# B&R Automation Studio project MIG1 (part 12)

```c
}
void readAttribute_CoolerSens(Arc_Link_typ *arc){
	// Create a Request Message and header
	Robot_typ *robot;
	Arc_Link_Request_typ *r;
	Arc_Link_Header_typ *h;
	PendingResponse_typ *pr;

	if(!arc) return;

	pr = &arc->PendingResponse;
	robot = &arc->robot;
	r = &arc->msgOUT.request;
	h = &arc->msgOUT.header;

	// Create a UDP Request Header with all the required info
	r->TimeoutTime = 10; // 10 ms
	r->Flags = 0;
	r->Retries = 1;
	r->MessageCounter = 0;
	r->AddressingMode = 6;
	r->ConnectionID = 15;
	r->MaximumObjs = 1;
	r->ServiceID.AttributeNumber = 0x7B09;
	r->ServiceID.StateNumber = 0;
	r->ServiceID.PropertyNumber = PROPERTY_ID_VALUE;

	//The attribute for the pump status (separate from the pump command) is 0x7875, and the attribute for the flow status is 0x7B09.

	r->SourceAddress = robot->arclink.network.ModuleBaseAddress;
	r->DestinationAddress = robot->miscSetup.CoolerAddr ;// Weld Controller
	r->Service = NETWORK_SERVICE_ATTRIBUTE_READ;
	r->MaxResponseSize = 254;

	//r->OutgoingData = er.encode();
	r->RequestSize = 0; // Size

	// Data must be sent in Big Endian format
	// Create a Response header for reply
	h->Flags 		= 0x02; // Arclink Request 0b0010

	// It has to be the same as request header
	h->Sequence 	= rand();
	pr->sqReadCoolerSens = h->Sequence;
	h->LastError 	= 0;
	h->DataLength 	= ARC_LINK_REQUEST_SIZE + r->RequestSize; // This depends on
	// size of data
	// being sent
	// 6(ARcklink
	// Response size +
	// Data size)

	/* Now encode ArcLink Header and Response */
	//arc->internal.OutMsgLen = ARC_LINK_HEADER_SIZE + h->DataLength;
	arc->internal.OutMsgLen = ARC_LINK_HEADER_SIZE + h->DataLength;

	// Temp Data
	int RequestSize = r->RequestSize;

	// Swap bytes into Big Endian Format
	swapArcLinkHeaderBytes(h);
	swapArcLinkRequestBytes(r);

	memcpy(arc->internal.pOutMsg, h , ARC_LINK_HEADER_SIZE);
	memcpy(arc->internal.pOutMsg + ARC_LINK_HEADER_SIZE, r , ARC_LINK_REQUEST_SIZE);

	// Swap bytes into Big Endian Format
	//swapArcLinkHeaderBytes(h);
	//swapArcLinkRequestBytes(r);

	// Arclink Request is ready to be sent
	writeMessageToOutgoingRingBuffer(arc);

	log_event(&robot->eventlog , "Get Cooler Sens REQ");
}

void action_ConfigDataSearch_GasSol(Arc_Link_typ *arc){
	// Create a Request Message and header
	Robot_typ *robot;
	Arc_Link_Request_typ *r;
	Arc_Link_Header_typ *h;
	PendingResponse_typ *pr;

	if(!arc) return;

	pr = &arc->PendingResponse;

	robot = &arc->robot;
	r = &arc->msgOUT.request;
	h = &arc->msgOUT.header;

	// Create a UDP Request Header with all the required info
	r->TimeoutTime = 10; // 10 ms
	r->Flags = 0;
	r->Retries = 1;
	r->MessageCounter = 0;
	r->AddressingMode = 6;
	r->ConnectionID = 15;
	r->MaximumObjs = 1;
	r->ServiceID.AttributeNumber = ACTION_CONFIG_DATA_SEARCH; //Configuration Data Search ACTION
	r->ServiceID.StateNumber = 0;
	r->ServiceID.PropertyNumber = PROPERTY_ID_VALUE;

	r->SourceAddress = robot->arclink.network.ModuleBaseAddress;
	r->DestinationAddress = WELD_CONTROLLER_NETWORK_ADDRESS; //BUS_MASTER_ARCLINK_NETWORK_ADDRESS;
	r->Service = NETWORK_SERVICE_ACTION;
	r->MaxResponseSize = 254;

	//r->OutgoingData = er.encode();
	r->RequestSize = 8; //
	USINT data[8];

	/*
	Request
	1 Byte	Search Parameter Mask
	1 Byte	Group Assignment
	2 Bytes Object Class
	1 Byte	Object Instance
	1 Byte	Object Class Type
	1 Byte	Maximum
	1 Byte	Starting Network Address
*/

	data[0] = 0x4; //Mask - Attribute Class

	data[1] = 0;

	data[2] = 0; //Bytes Object Class
	//data[3] = 29; //Bytes Object Class - Cooler
	data[3] = 22; //Bytes Object Class - Remote Control object (object class ID 22)

	data[4] = 0;
	data[5] = 0;
	data[6] = 1;
	data[7] = 1;

	memcpy(arc->internal.pOutMsg + ARC_LINK_HEADER_SIZE + ARC_LINK_REQUEST_SIZE, &data[0] , r->RequestSize);

	// Data must be sent in Big Endian format
	// Create a Response header for reply
	h->Flags 		= 0x02; // Arclink Request 0b0010

	// It has to be the same as request header
	h->Sequence 	= rand();
	h->LastError 	= 0;
	h->DataLength 	= ARC_LINK_REQUEST_SIZE + r->RequestSize; // This depends on
	// size of data
	// being sent
	// 6(ARcklink
	// Response size +
	// Data size)

	/* Now encode ArcLink Header and Response */
	//arc->internal.OutMsgLen = ARC_LINK_HEADER_SIZE + h->DataLength;
	arc->internal.OutMsgLen = ARC_LINK_HEADER_SIZE + h->DataLength;

	pr->sqConfigDataSearchAction_GasSol = 	h->Sequence;

	// Temp Data
	int RequestSize = r->RequestSize;

	// Swap bytes into Big Endian Format
	swapArcLinkHeaderBytes(h);
	swapArcLinkRequestBytes(r);

	memcpy(arc->internal.pOutMsg, h , ARC_LINK_HEADER_SIZE);
	memcpy(arc->internal.pOutMsg + ARC_LINK_HEADER_SIZE, r , ARC_LINK_REQUEST_SIZE);

	// Swap bytes into Big Endian Format
	//swapArcLinkHeaderBytes(h);
	//swapArcLinkRequestBytes(r);

	// Arclink Request is ready to be sent

	writeMessageToOutgoingRingBuffer(arc);

	log_event(&robot->eventlog , "Get Cooler Adr REQ");
}

void action_ConfigDataSearch(Arc_Link_typ *arc){
	// Create a Request Message and header
	Robot_typ *robot;
	Arc_Link_Request_typ *r;
	Arc_Link_Header_typ *h;
	PendingResponse_typ *pr;

	if(!arc) return;

	pr = &arc->PendingResponse;

	robot = &arc->robot;
	r = &arc->msgOUT.request;
	h = &arc->msgOUT.header;

	// Create a UDP Request Header with all the required info
	r->TimeoutTime = 10; // 10 ms
	r->Flags = 0;
	r->Retries = 1;
	r->MessageCounter = 0;
	r->AddressingMode = 6;
	r->ConnectionID = 15;
	r->MaximumObjs = 1;
	r->ServiceID.AttributeNumber = ACTION_CONFIG_DATA_SEARCH; //Configuration Data Search ACTION
	r->ServiceID.StateNumber = 0;
	r->ServiceID.PropertyNumber = PROPERTY_ID_VALUE;

	r->SourceAddress = robot->arclink.network.ModuleBaseAddress;
	r->DestinationAddress = WELD_CONTROLLER_NETWORK_ADDRESS; //BUS_MASTER_ARCLINK_NETWORK_ADDRESS;
	r->Service = NETWORK_SERVICE_ACTION;
	r->MaxResponseSize = 254;

	//r->OutgoingData = er.encode();
	r->RequestSize = 8; //
	USINT data[8];

	/*
	Request
	1 Byte	Search Parameter Mask
	1 Byte	Group Assignment
	2 Bytes Object Class
	1 Byte	Object Instance
	1 Byte	Object Class Type
	1 Byte	Maximum
	1 Byte	Starting Network Address
*/

	data[0] = 0x4; //Mask - Attribute Class

	data[1] = 0;

	data[2] = 0; //Bytes Object Class
	data[3] = 29; //Bytes Object Class - Cooler
	//data[3] = 22; //Bytes Object Class - Remote Control object (object class ID 22)

	data[4] = 0;
	data[5] = 0;
	data[6] = 1;
	data[7] = 1;

	memcpy(arc->internal.pOutMsg + ARC_LINK_HEADER_SIZE + ARC_LINK_REQUEST_SIZE, &data[0] , r->RequestSize);

	// Data must be sent in Big Endian format
	// Create a Response header for reply
	h->Flags 		= 0x02; // Arclink Request 0b0010

	// It has to be the same as request header
	h->Sequence 	= rand();
	h->LastError 	= 0;
	h->DataLength 	= ARC_LINK_REQUEST_SIZE + r->RequestSize; // This depends on
	// size of data
	// being sent
	// 6(ARcklink
	// Response size +
	// Data size)

	/* Now encode ArcLink Header and Response */
	//arc->internal.OutMsgLen = ARC_LINK_HEADER_SIZE + h->DataLength;
	arc->internal.OutMsgLen = ARC_LINK_HEADER_SIZE + h->DataLength;

	pr->sqConfigDataSearchAction = 	h->Sequence;

	// Temp Data
	int RequestSize = r->RequestSize;

	// Swap bytes into Big Endian Format
	swapArcLinkHeaderBytes(h);
	swapArcLinkRequestBytes(r);

	memcpy(arc->internal.pOutMsg, h , ARC_LINK_HEADER_SIZE);
	memcpy(arc->internal.pOutMsg + ARC_LINK_HEADER_SIZE, r , ARC_LINK_REQUEST_SIZE);

	// Swap bytes into Big Endian Format
	//swapArcLinkHeaderBytes(h);
	//swapArcLinkRequestBytes(r);

	// Arclink Request is ready to be sent

	writeMessageToOutgoingRingBuffer(arc);

	log_event(&robot->eventlog , "Get Cooler Adr REQ");
}

void handleResponse_ReadCoolerSens(Arc_Link_typ *arc){
	Arc_Link_Response_typ 	*r; // temp reference to request
	Robot_typ 				*robot;
	USINT *data;

	if (!arc) return; // Prevent null pointer reference
	r = &arc->msgIN.response;
	robot = &arc->robot;

	DBG_OB("Received response for Cooler Search Address \r\n" );

	//Log.d(TAG, "Recevied Assign Network Address Action");

	// Copy Data if available to the Incoming data pointer
	if(r->ResponseSize > 0){
		//byte[] data = r.OutgoingData; // incominng data in Big endian format
		data = (arc->internal.pInMsg + ARC_LINK_HEADER_SIZE + ARC_LINK_RESPONSE_SIZE); // Pointer to data go back here and test
	}else{
		DBG_OB("Error: Receiving fault status with Response size \r\n");
		log_error(&robot->errorlog , "Cooler Sens Resp Fault");
		return;
	}

	//robot->miscSetup.CoolerAddr = data[0];
	//log_event(&robot->eventlog , "Got Cooler Adr RESP");

	robot->Cntrl.Fbk.coolerSens_Status = data[0];
	log_event(&robot->eventlog , "Got Cooler Sens");

}

void handleResponseReadControlParamDataAction(Arc_Link_typ *arc){
	Arc_Link_Response_typ 	*r; // temp reference to request
	Robot_typ 				*robot;
	USINT *data;

	if (!arc) return; // Prevent null pointer reference
	r = &arc->msgIN.response;
	robot = &arc->robot;

	DBG_OB("Received response -Read WC Param Data Action\r\n" );
	//log_event(&robot->eventlog , "Received Cooler Address from PS");

	//Log.d(TAG, "Recevied Assign Network Address Action");

	// Copy Data if available to the Incoming data pointer
	if(r->ResponseSize > 0){
		//byte[] data = r.OutgoingData; // incominng data in Big endian format
		data = (arc->internal.pInMsg + ARC_LINK_HEADER_SIZE + ARC_LINK_RESPONSE_SIZE); // Pointer to data go back here and test
		log_event(&robot->eventlog , "Got WC Param Data");
	}else{
		//DBG_OB("Error: Receiving fault status with Response size \r\n");
		log_error(&robot->errorlog , "Get WC Param Data Fault");
		return;
	}

	memset (&robot->Comm.CntrlParamData , 0 , sizeof(ReadControlParameterData_typ));
	memset (&robot->ResData_raw , 0 , sizeof(robot->ResData_raw));
	robot->ResDataSize = 0;

	if(r->ResponseSize == 1){ // return code

		robot->Comm.CntrlParamData.ReturnCode = *data;
	}
	else if((r->ResponseSize > 0)
		&&(r->ResponseSize < 32)){
		robot->ResDataSize = (UINT)r->ResponseSize;
		memcpy(robot->ResData_raw , data , r->ResponseSize);
	}
	else
		return;

	memcpy(&robot->Comm.CntrlParamData.MaxVal , (data+0) , 2);
	swapBytes((USINT *)&robot->Comm.CntrlParamData.MaxVal, 2);

	memcpy(&robot->Comm.CntrlParamData.MinVal , (data +2) , 2);
	swapBytes((USINT *)&robot->Comm.CntrlParamData.MinVal, 2);

	robot->Comm.CntrlParamData.UnitsCode = (USINT)*(data+4);

	robot->Comm.CntrlParamData.DecimalPlace = (USINT)*(data+5);
	memcpy(robot->Comm.CntrlParamData.Name ,  data+6 , 17);
	//swapBytes(robot->Comm.CntrlParamData.Name, 17);

}

void handleResponseConfigDataSearchAction_GasSol(Arc_Link_typ *arc){
	Arc_Link_Response_typ 	*r; // temp reference to request
	Robot_typ 				*robot;
	USINT *data;

	if (!arc) return; // Prevent null pointer reference
	r = &arc->msgIN.response;
	robot = &arc->robot;

	DBG_OB("Received response for Cooler Search Address \r\n" );
	//log_event(&robot->eventlog , "Received Cooler Address from PS");

	//Log.d(TAG, "Recevied Assign Network Address Action");

	// Copy Data if available to the Incoming data pointer
	if(r->ResponseSize > 0){
		//byte[] data = r.OutgoingData; // incominng data in Big endian format
		data = (arc->internal.pInMsg + ARC_LINK_HEADER_SIZE + ARC_LINK_RESPONSE_SIZE); // Pointer to data go back here and test
	}else{
		DBG_OB("Error: Receiving fault status with Response size \r\n");
		log_error(&robot->errorlog , "Gas Sol Addr Fault");
		return;
	}

	robot->miscSetup.GasSolAddr = data[0];
	log_event(&robot->eventlog , "Got Gas Sol Adr RESP");

}

void handleResponseConfigDataSearchAction(Arc_Link_typ *arc){
	Arc_Link_Response_typ 	*r; // temp reference to request
	Robot_typ 				*robot;
	USINT *data;

	if (!arc) return; // Prevent null pointer reference
	r = &arc->msgIN.response;
	robot = &arc->robot;

	DBG_OB("Received response for Cooler Search Address \r\n" );
	//log_event(&robot->eventlog , "Received Cooler Address from PS");

	//Log.d(TAG, "Recevied Assign Network Address Action");

	// Copy Data if available to the Incoming data pointer
	if(r->ResponseSize > 0){
		//byte[] data = r.OutgoingData; // incominng data in Big endian format
		data = (arc->internal.pInMsg + ARC_LINK_HEADER_SIZE + ARC_LINK_RESPONSE_SIZE); // Pointer to data go back here and test
	}else{
		DBG_OB("Error: Receiving fault status with Response size \r\n");
		log_error(&robot->errorlog , "Cooler Addr Fault");
		return;
	}

	robot->miscSetup.CoolerAddr = data[0];
	log_event(&robot->eventlog , "Got Cooler Adr RESP");

}

/*
	Error Logger by Obed Rev 1.0
*/
void log_error(Log_typ* err, char* msg){
	if(!err) return;

	// Healthy Inialization
	if(!err->pLog){
		err->pLog = &err->log;
	}

	memmove((void *)(err->pLog + LOG_MAX_LENGTH), (void *)err->pLog, (LOG_MAX_LENGTH * (LOG_MAX_LINE - 1) ));
	memmove( (void *)(err->pLog), (void *)msg, (LOG_MAX_LENGTH) );
}

void log_event(Log_typ* event, char* msg){
	if(!event) return;

	// Healthy Inialization
	if(!event->pLog){
		event->pLog = &event->log;
	}

	memmove((void *)(event->pLog + LOG_MAX_LENGTH), (void *)event->pLog, (LOG_MAX_LENGTH * (LOG_MAX_LINE - 1) ));
	memmove( (void *)(event->pLog), (void *)msg, (LOG_MAX_LENGTH) );
}
```

### Robot.c
```c
/*
 * Handler.c
 *
 *  Created on: May 18, 2017
 *      Author: Obed Bardales
 */
#ifndef _ROBOT_C
#define _ROBOT_C

/* Handle Robot Cyclic Operations */
void handleRobotCyclicOps(Arc_Link_typ *arc){
	if(!arc) return;

	// Handle Mr.Robot interface
	handleRobotInterface(arc);

	// "The difference is not one thing, it's everything!"
}

/* Get Network Configuration from Robot */
void getNetworkConfigurationAttribute(Arc_Link_typ *arc, USINT *ResponseData){
	Arc_Link_Request_typ *req;
	Arc_Link_Response_typ *r;
	Robot_typ *robot;
	ServiceID_typ *serviceID;
	ArcLinkObject_typ *arclink;
	USINT data[10]; // Temp Data place holder
	UINT txtlength; // text length

	if(!arc) return;
	if(!ResponseData) return;

	robot = &arc->robot; // Reference to Robot
	req = &arc->msgIN.request;
	serviceID = &req->ServiceID;
	r = &arc->msgOUT.response;
	arclink = &robot->arclink;
	int dataSize = req->MaxResponseSize;

	/* Attribute Number */
	switch (serviceID->AttributeNumber) {

		case VENDOR_ID: /* 0 */
			// MaxDataSize = 2
			// Big Endian Format

			data[0] = (USINT) (arclink->network.VendorID >> 8);
			data[1] = (USINT) (arclink->network.VendorID >> 0);
			memcpy(ResponseData, data, 2);
			r->ResponseSize = 2;

			return;

		case CLASS_ID: /* 4 */
			// MaxDataSize = 2
			// Big Endian Format
			data[0] = (USINT) (arclink->network.ClassID >> 8);
			data[1] = (USINT) (arclink->network.ClassID >> 0);
			memcpy(ResponseData, data, 2);
			r->ResponseSize = 2;
			return;

		case CLASS_TYPE: /* 7 */
			// MaxDataSize = 2
			// Big Endian Format
			data[0] = (USINT) (arclink->network.ClassType >> 0);
			memcpy(ResponseData, data, 1);
			r->ResponseSize = 1;
			return;

		case GROUP_ASSIGNMENTS: /* 10 */
			// MaxDataSize = 2
			// Big Endian Format
			data[0] = (USINT) (arclink->network.GroupAssignments >> 0);
			memcpy(ResponseData, data, 1);
			r->ResponseSize = 1;
			return;

		case INSTANCE_ASSIGNMENTS: /* 11 */
			// MaxDataSize = 2
			// Big Endian Format
			data[0] = (USINT) (arclink->network.InstanceAssignments >> 0);
			memcpy(ResponseData, data, 1);
			r->ResponseSize = 1;
			return;

		case FAULT_STATUS: /* 14 */
			// MaxDataSize = 2
			// Big Endian Format
			data[0] = (USINT) (arclink->network.FaultStatus >> 0);
			memcpy(ResponseData, data, 1);
			r->ResponseSize = 1;
			return;

		case SILICON_SERIAL_NUMBER: /* 16 */
			// MaxDataSize = 2
			// Big Endian Format
			data[0] = (USINT) (arclink->network.SiliconSerialNumber >> 8);
			data[1] = (USINT) (arclink->network.SiliconSerialNumber >> 0);
			memcpy(ResponseData, data, 2);
			r->ResponseSize = 2;
			return;

		case NUMBER_OF_EMBEDDED_OBJECTS: /* 17 */
			// MaxDataSize = 2
			// Big Endian Format
			data[0] = (USINT) (arclink->network.NumberofEmbeddedObjects >> 0);
			memcpy(ResponseData, data, 1);
			r->ResponseSize = 1;
			return;

		case SOFTWARE_VERSION: /* 19 */
			// MaxDataSize = 64
			// Big Endian Format
			txtlength = strlen(arclink->network.SoftwareVersion);
			// Swap Bytes before sendSuccesfullWriteAttributeConfirmation
			//swapBytes(arclink->network.SoftwareVersion, txtlength);
			memcpy(ResponseData, arclink->network.SoftwareVersion, txtlength);
			//swapBytes(arclink->network.SoftwareVersion, txtlength);
			r->ResponseSize = txtlength;
			return;

		case BOOTSTRAP: /* 24 */
			// MaxDataSize = 2
			// Big Endian Format
			data[0] = (USINT) (arclink->network.Bootstrap >> 0);
			memcpy(ResponseData, data, 1);
			r->ResponseSize = 1;
			return;

		case PAIRED_ITEMS_COUNT: /* 50 */
			// MaxDataSize = 2
			// Big Endia Format
			data[0] = (USINT) (arclink->network.PairedItemsCount >> 8);
			data[1] = (USINT) (arclink->network.PairedItemsCount >> 0);
			memcpy(ResponseData, data, 2);
			r->ResponseSize = 2;
			return;
	}
}

/* Write Network Configuration Attribute */
BOOL writeNetworkConfigurationAttribute(Arc_Link_typ *arc){

	BOOL success = 1;

	UINT *data;

	Arc_Link_Request_typ *req;
	ServiceID_typ *serviceID;
	Robot_typ *robot;
	ArcLinkObject_typ *arclink;
	if(!arc) return;

	req = &arc->msgIN.request;
	serviceID = &req->ServiceID;
	robot = &arc->robot;
	arclink = &robot->arclink;

	DBG("Inside writeNetworkConfigurationAttribute \r\n" );
	//Log.d(TAG, "Recevied Assign Network Address Action");

	// Copy Data if available to the Incoming data pointer
	if(req->RequestSize > 0){
	//byte[] data = r.OutgoingData; // incominng data in Big endian format
		data = (arc->internal.pInMsg + ARC_LINK_HEADER_SIZE + ARC_LINK_REQUEST_SIZE); // Pointer to data
	}else{
		DBG("Error: writeNetworkConfigurationAttribute, Error with Request size\r\n" );
		return;
	}

	/* Attribute Number */
	switch (serviceID->AttributeNumber) {

	// Currently Supported Attributes by the Robot
	case RESET:
		arclink->network.Reset = *(data + 0);//data[0]; // Size is typically 1 byte
		arclink->network.BusAvailable = 0; // Robot must enter to unmapped state
		robot->isMapping = 0;
		robot->isMapped = 0;
		robot->Cntrl.Fbk.Status &= ~ArcLink_Mapped;
		robot->Cntrl.Fbk.Status &= ~ArcLink_Mapping;
		robot->isMiscSetupOneShot = 0;
		DBG("Setting Robot to Unmapped state\r\n" );
		break;

	case GROUP_ASSIGNMENTS:
		arclink->network.GroupAssignments = *(data + 0);///data[0]; // Size is typically 1
													// byte

		break;

	case INSTANCE_ASSIGNMENTS:
		arclink->network.InstanceAssignments = *(data + 0);///data[0]; // Size is typically
														// 1 byte
		break;

	case BUS_AVAILABLE:
		arclink->network.BusAvailable = *(data + 0); //data[0]; // Size is typically 1 byte
		robot->isMapping 	= 0;
		robot->isMapped 	= 1;
		robot->Cntrl.Fbk.Status |= ArcLink_Mapped;
		robot->Cntrl.Fbk.Status &= ~ArcLink_Mapping;
		DBG("Robot was mapped succesfully Świetny programista! \r\n" );
		log_event(&robot->eventlog , "Arc Link Mapped");
		break;

	}

	return success; // Whether Attribute was written succesfully

}

void handleRobotInterface(Arc_Link_typ *arc){

	Robot_typ *robot;
	Robot_Intrf_typ *intrf;
	if(!arc) return;

	robot = &arc->robot;
	intrf = &robot->Intrf;

	// Robot must be Mapped with WeldController
	if(!robot->isMapped) return;

	//  Handle state changes from outside and provide feedback

	handleRobotCntrl(arc);
	error_status_handler(arc);
	ArcLink_Timer(arc);
	/////////

	// Handle xCMD
	switch(intrf->xCMD) {
		/* Turn Power Supply ON */
		case ROBOT_CMD_PS_ON:
			writeOutputOnCommand(arc);
			DBG("Robot commanded Power Supply ON! \r\n" );
			log_event(&robot->eventlog , "PS ON Cmd");
			break;

		/* Turn Power Supply OFF */
		case ROBOT_CMD_PS_OFF:
			writeOutputOffCommand(arc);
			DBG("Robot commanded Power Supply OFF! \r\n" );
			log_event(&robot->eventlog , "PS OFF Cmd");
			break;

		/* Set Controls Action Request */
		case ROBOT_SET_CONTROLS:
			createSetControlsAction(arc);
			DBG("Robot sent Set Controls Action Request! \r\n" );
			break;

		case ROBOT_CMD_COOLER_ON:
			writeOutputCoolerOnCommand(arc);
			DBG("Robot commanded Cooler ON! \r\n" );

		break;

		case ROBOT_CMD_COOLER_OFF:
			writeOutputCoolerOffCommand(arc);
			DBG("Robot commanded Cooler OFF! \r\n" );

		break;

		case ROBOT_CMD_SEARCH_COOLER_ADR:
			action_ConfigDataSearch(arc);
			DBG("commanded Get Cooler Adr! \r\n" );
		break;

		case ROBOT_READ_COOLER_SENS:
			readAttribute_CoolerSens(arc);
			DBG("commanded Get Cooler Sens! \r\n" );
		break;

		case ROBOT_READ_WC_PARAM_DATA:
			createReadCntrlParamDataAction(arc);
			DBG("commanded Read WC Param Data! \r\n" );
		break;

		case ROBOT_CMD_SEARCH_GAS_SOL_ADR:
			action_ConfigDataSearch_GasSol(arc);
			DBG("commanded Get Gas Sol  Adr! \r\n" );
		break;

		case ROBOT_CMD_GAS_SOL_ENABLE: // Make  Gas Sol “Manual Valve”

			writeOutputGasEnableCommand(arc);
			DBG("Robot commanded Gas Enable\r\n" );

		break;

		case ROBOT_CMD_GAS_SOL_ON: // Turn On Gas Sol

			writeOutputGasOnCommand(arc);
			DBG("Robot commanded Gas ON\r\n" );

		break;

		case ROBOT_CMD_GAS_SOL_OFF:	// Turn Off Gas Sol

			writeOutputGasOffCommand(arc);
			DBG("Robot commanded Gas OFF\r\n" );

		break;

	}

	// Clear xCMD
	if (intrf->xCMD > 0) intrf->xCMD = 0;

}

void handleRobotCntrl(Arc_Link_typ *arc){

	Robot_typ *robot;
	Robot_Intrf_typ *intrf;
	if(!arc) return;

	robot = &arc->robot;
	intrf = &robot->Intrf;

	//*************** CMD  *****************************/
	//**************Highest priority CMD****************//
	if(robot->Cntrl.Cmd.COOLER && !robot->Cntrl.Int._COOLER){

		intrf->xCMD = ROBOT_CMD_COOLER_ON;
		robot->Cntrl.Int._COOLER  = robot->Cntrl.Cmd.COOLER;

	}
	else if(robot->Cntrl.Cmd.RUN != robot->Cntrl.Int._RUN){

		if(robot->Cntrl.Cmd.RUN)
			intrf->xCMD = ROBOT_CMD_PS_ON;
		else
			intrf->xCMD = ROBOT_CMD_PS_OFF;

		robot->Cntrl.Int._RUN  = robot->Cntrl.Cmd.RUN;
	}
	else if(!robot->Cntrl.Cmd.COOLER && robot->Cntrl.Int._COOLER){

		intrf->xCMD = ROBOT_CMD_COOLER_OFF;
		robot->Cntrl.Int._COOLER  = robot->Cntrl.Cmd.COOLER;

	}
	//robot->Cntrl.Int._RUN  = robot->Cntrl.Cmd.RUN;
	//robot->Cntrl.Int._COOLER  = robot->Cntrl.Cmd.COOLER;

	//********************************************************//

	if(!intrf->xCMD){

		/*
		1 Byte	Parameter Mask
		2 Bytes	Weld Mode 	If parameter mask bit 0 set.
		2 Bytes	Work-point	If parameter mask bit 1 set.
		2 Bytes	Trim	If parameter mask bit 2 set.
		2 Bytes	Wave-Control 1	If parameter mask bit 3 set.
		2 Bytes	Wave-Control 2	If parameter mask bit 4 set.
		2 Bytes	Wave-Control 3	If parameter mask bit 5 set.
		2 Bytes	Wave-Control 4	If parameter mask bit 6 set.
		*/

		switch(robot->Cntrl.Cmd.Mode){

			case 3:

				if((robot->Cntrl.Cmd.Mode != robot->Cntrl.Int._Mode )
					|| (robot->Cntrl.Cmd.AmpSP != robot->Cntrl.Int._AmpSP )
					|| (robot->Cntrl.Cmd.BckAmpSP != robot->Cntrl.Int._BckAmpSP )
					|| (robot->Cntrl.Cmd.PulseFreq != robot->Cntrl.Int._PulseFreq )
					|| (robot->Cntrl.Cmd.PulseWidth != robot->Cntrl.Int._PulseWidth )){

					robot->wc.setup.ctrlParam.ParameterMask = 0x23; // 0b0100011; // change accordingly for Mode 3
					UINT *mode 	= &robot->Cntrl.Cmd.Mode; // Mode
					UINT ampSP = (UINT)robot->Cntrl.Cmd.AmpSP; //amps
					robot->wc.setup.ctrlParam.WeldMode = *mode;
					robot->wc.setup.ctrlParam.WorkPoint = ampSP;
					robot->wc.setup.ctrlParam.WaveControl3 = 1; // Hot pulse. Need info from Lincoln

					// This command write Controls Parameter into Power Supply
					intrf->xCMD = ROBOT_SET_CONTROLS;

				}

				robot->Cntrl.Int._Mode 			= robot->Cntrl.Cmd.Mode;
				robot->Cntrl.Int._AmpSP 		= robot->Cntrl.Cmd.AmpSP;
				robot->Cntrl.Int._BckAmpSP 		= robot->Cntrl.Cmd.BckAmpSP;
				robot->Cntrl.Int._PulseFreq 	= robot->Cntrl.Cmd.PulseFreq;
				robot->Cntrl.Int._PulseWidth 	= robot->Cntrl.Cmd.PulseWidth;

			break;

			case 5:

				if((robot->Cntrl.Cmd.Mode != robot->Cntrl.Int._Mode )
					|| (robot->Cntrl.Cmd.Volts != robot->Cntrl.Int._Volts )
					|| (robot->Cntrl.Cmd.Pinch != robot->Cntrl.Int._Pinch )
					){

					robot->wc.setup.ctrlParam.ParameterMask = 0x0D; // 0b0001011; // change accordingly for Mode 5
					UINT *mode 	= &robot->Cntrl.Cmd.Mode; // Mode
					UINT VoltsSP = (UINT)(robot->Cntrl.Cmd.Volts * 10); //Volts
					robot->wc.setup.ctrlParam.WeldMode = *mode;
					robot->wc.setup.ctrlParam.WorkPoint = VoltsSP;
					robot->wc.setup.ctrlParam.WaveControl1 = (UINT)(robot->Cntrl.Cmd.Pinch * 10);

					// This command write Controls Parameter into Power Supply
					intrf->xCMD = ROBOT_SET_CONTROLS;

				}

				robot->Cntrl.Int._Mode 			= robot->Cntrl.Cmd.Mode;
				robot->Cntrl.Int._Volts 		= robot->Cntrl.Cmd.Volts;
				robot->Cntrl.Int._Pinch 		= robot->Cntrl.Cmd.Pinch;

			break;

			case 21:

				if((robot->Cntrl.Cmd.Mode != robot->Cntrl.Int._Mode )
					|| (robot->Cntrl.Cmd.WFS != robot->Cntrl.Int._WFS)
					|| (robot->Cntrl.Cmd.Volts != robot->Cntrl.Int._Volts )
					|| (robot->Cntrl.Cmd.Pinch != robot->Cntrl.Int._Pinch )
					|| robot->Cntrl.Cmd.SendParam
					){

					robot->Cntrl.Cmd.SendParam = 0;

					robot->wc.setup.ctrlParam.ParameterMask = 0x0F; // 0b0001111; // change accordingly for Mode 5
					UINT *mode 	= &robot->Cntrl.Cmd.Mode; // Mode
					UINT WFS_SP = (UINT)(robot->Cntrl.Cmd.WFS * 1); //WF
					UINT VoltsSP = (UINT)(robot->Cntrl.Cmd.Volts * 10); //Volts
					UINT PinchSP = (UINT)(robot->Cntrl.Cmd.Pinch * 10); //Pinch

					if(robot->Cntrl.Cmd.Development)
						robot->wc.setup.ctrlParam.WeldMode = 0;
					else
						robot->wc.setup.ctrlParam.WeldMode = *mode;

					robot->wc.setup.ctrlParam.WorkPoint = WFS_SP;
					robot->wc.setup.ctrlParam.Trim = VoltsSP;
					robot->wc.setup.ctrlParam.WaveControl1 = PinchSP;

					// This command write Controls Parameter into Power Supply
					intrf->xCMD = ROBOT_SET_CONTROLS;

					robot->Cntrl.Int._Mode 			= robot->Cntrl.Cmd.Mode;
					robot->Cntrl.Int._WFS 			= robot->Cntrl.Cmd.WFS;
					robot->Cntrl.Int._Volts 		= robot->Cntrl.Cmd.Volts;
					robot->Cntrl.Int._Pinch 		= robot->Cntrl.Cmd.Pinch;

				}

			break;

			case 22:

				if((robot->Cntrl.Cmd.Mode != robot->Cntrl.Int._Mode )
					|| (robot->Cntrl.Cmd.WFS != robot->Cntrl.Int._WFS)
					|| (robot->Cntrl.Cmd.Trim != robot->Cntrl.Int._Trim )
					|| (robot->Cntrl.Cmd.UltimArc != robot->Cntrl.Int._UltimArc )
					|| robot->Cntrl.Cmd.SendParam
					){

					robot->Cntrl.Cmd.SendParam = 0;

					robot->wc.setup.ctrlParam.ParameterMask = 0x0F; // 0b0001111; // change accordingly for Mode 5
					UINT *mode 	= &robot->Cntrl.Cmd.Mode; // Mode
					UINT WFS_SP = (UINT)(robot->Cntrl.Cmd.WFS * 1); // WF
					UINT TrimSP = (UINT)(robot->Cntrl.Cmd.Trim * 100); // Trim
					UINT UltimArcSP = (UINT)(robot->Cntrl.Cmd.UltimArc * 10); //Pinch

					if(robot->Cntrl.Cmd.Development)
						robot->wc.setup.ctrlParam.WeldMode = 0;
					else
						robot->wc.setup.ctrlParam.WeldMode = *mode;

					robot->wc.setup.ctrlParam.WorkPoint = WFS_SP;
					robot->wc.setup.ctrlParam.Trim = TrimSP;
					robot->wc.setup.ctrlParam.WaveControl1 = UltimArcSP;

					// This command write Controls Parameter into Power Supply
					intrf->xCMD = ROBOT_SET_CONTROLS;

					robot->Cntrl.Int._Mode 			= robot->Cntrl.Cmd.Mode;
					robot->Cntrl.Int._WFS 			= robot->Cntrl.Cmd.WFS;
					robot->Cntrl.Int._Trim 			= robot->Cntrl.Cmd.Trim;
					robot->Cntrl.Int._UltimArc 		= robot->Cntrl.Cmd.UltimArc;

				}

			break;

			case 160:
			case 161:
			case 162:
			case 163:
			case 164:
			case 165:
			case 166:
			case 167:

				if((robot->Cntrl.Cmd.Mode != robot->Cntrl.Int._Mode )
					|| (robot->Cntrl.Cmd.Volts != robot->Cntrl.Int._Volts )
					//|| (robot->Cntrl.Cmd.Pinch != robot->Cntrl.Int._Pinch )
					){

					robot->wc.setup.ctrlParam.ParameterMask = 0x03; // 0b0000011; // Volts and WaveCntr 1

					//robot->wc.setup.ctrlParam.ParameterMask = 0x01; // Only Volts

					UINT *mode 	= &robot->Cntrl.Cmd.Mode; // Mode
					UINT VoltsSP = (UINT)(robot->Cntrl.Cmd.Volts * 10); // Volts
					robot->wc.setup.ctrlParam.WeldMode = *mode;
					robot->wc.setup.ctrlParam.WorkPoint = VoltsSP;
					//robot->wc.setup.ctrlParam.WaveControl1 = (UINT)(robot->Cntrl.Cmd.Pinch * 10);
					robot->wc.setup.ctrlParam.WaveControl1 = 0;

					// This command write Controls Parameter into Power Supply
					intrf->xCMD = ROBOT_SET_CONTROLS;

				}

				robot->Cntrl.Int._Mode 			= robot->Cntrl.Cmd.Mode;
				robot->Cntrl.Int._Volts 		= robot->Cntrl.Cmd.Volts;
				//robot->Cntrl.Int._Pinch 		= robot->Cntrl.Cmd.Pinch;

			break;

			case 170:

				if((robot->Cntrl.Cmd.Mode != robot->Cntrl.Int._Mode )
					|| (robot->Cntrl.Cmd.WFS != robot->Cntrl.Int._WFS)
					|| (robot->Cntrl.Cmd.Volts != robot->Cntrl.Int._Volts )
					|| (robot->Cntrl.Cmd.UltimArc != robot->Cntrl.Int._UltimArc )
					|| robot->Cntrl.Cmd.SendParam
					){

					robot->Cntrl.Cmd.SendParam = 0;

					robot->wc.setup.ctrlParam.ParameterMask = 0x0F; // 0b0001111; // change accordingly for Mode 5
					UINT *mode 	= &robot->Cntrl.Cmd.Mode; // Mode
					UINT WFS_SP = (UINT)(robot->Cntrl.Cmd.WFS * 1); //WF
					UINT VoltsSP = (UINT)(robot->Cntrl.Cmd.Volts * 10); //Volts
					UINT UltimArcSP = (UINT)(robot->Cntrl.Cmd.UltimArc * 10); //UltimArc

					if(robot->Cntrl.Cmd.Development)
						robot->wc.setup.ctrlParam.WeldMode = 0;
					else
						robot->wc.setup.ctrlParam.WeldMode = *mode;

					robot->wc.setup.ctrlParam.WorkPoint = WFS_SP;
					robot->wc.setup.ctrlParam.Trim = VoltsSP;
					robot->wc.setup.ctrlParam.WaveControl1 = UltimArcSP;

					// This command write Controls Parameter into Power Supply
					intrf->xCMD = ROBOT_SET_CONTROLS;

					robot->Cntrl.Int._Mode 			= robot->Cntrl.Cmd.Mode;
					robot->Cntrl.Int._WFS 			= robot->Cntrl.Cmd.WFS;
					robot->Cntrl.Int._Volts 		= robot->Cntrl.Cmd.Volts;
					robot->Cntrl.Int._UltimArc 		= robot->Cntrl.Cmd.UltimArc;

				}

			break;

			case 200:  // Calibration Current

				if((robot->Cntrl.Cmd.Mode != robot->Cntrl.Int._Mode )
					|| (robot->Cntrl.Cmd.AmpSP != robot->Cntrl.Int._AmpSP )
					){

					robot->wc.setup.ctrlParam.ParameterMask = 0x03; // 0b0000011; // change accordingly for Mode 200
					UINT *mode 	= &robot->Cntrl.Cmd.Mode; // Mode
					UINT AmpSP = (UINT)(robot->Cntrl.Cmd.AmpSP * 1); //amps
					robot->wc.setup.ctrlParam.WeldMode = *mode;
					robot->wc.setup.ctrlParam.WorkPoint = AmpSP;

					// This command write Controls Parameter into Power Supply
					intrf->xCMD = ROBOT_SET_CONTROLS;

				}

				robot->Cntrl.Int._Mode 			= robot->Cntrl.Cmd.Mode;
				robot->Cntrl.Int._AmpSP 		= robot->Cntrl.Cmd.AmpSP;

			break;

		}

	}
	//********************************************************//

	//*****************Lowest Priority CMD ********************//
	if(!intrf->xCMD){
		if(robot->Cntrl.Cmd.RST != robot->Cntrl.Int._RST){

			robot->Cntrl.Fbk.Status = 0;
			robot->miscSetup.state = 0; //reset misc state machine state
			robot->miscSetup.CoolerAddr = 0;
			robot->isMapping = 0;
			robot->isMapped = 0;	    //clear flag, set to unmapped status, stop timer
			robot->isMiscSetupOneShot = 0;
			robot->Comm.ArcComTimer.IN = 0;
			robot->Comm.StopRespondHeartBeat = 1; //halt heartbeat,force master to send out RESET request

		}
		robot->Cntrl.Int._RST 			= robot->Cntrl.Cmd.RST;

	}

	//*************** FEEDBACK  *****************************/

	robot->Cntrl.Fbk.curArcVolt = robot->wc.data.telemetry.fVoltage;
	robot->Cntrl.Fbk.curArcAmp  = robot->wc.data.telemetry.fCurrent;
	//robot->Cntrl.Fbk.Error      =  ???????
	//robot->Cntrl.Fbk.Status      =  ???????

	//********************************************************//

	return;

}

void error_status_handler(Arc_Link_typ *arc)
{

	Robot_typ *robot;
	if(!arc) return;

	robot = &arc->robot;

	// System is ready when mapped, ready status from PS is set and Arc Link Active, could add no system fault here
	if ((robot->isReady) && (robot->isMapped) && (robot->Comm.ArcLinkActive) && !robot->Cntrl.Fbk.Error)
	{
		robot->Cntrl.Fbk.Status |= PS_Ready;
//		log_event(&robot->eventlog , "Power supply is ready");
	}

	else
		robot->Cntrl.Fbk.Status &= ~PS_Ready;

	/*
	if ((robot->Cntrl.Fbk.Error >> 1 & 0x0001) || (robot->Cntrl.Fbk.Error >> 2 & 0x0001))  //either system fault from PS or network error will generate fault condition
		robot->Cntrl.Fbk.Error |= PS_Error_Present;
	else
		robot->Cntrl.Fbk.Error &= ~PS_Error_Present;
	*/
}
void ArcLink_Timer(Arc_Link_typ *arc){
//
	Robot_typ *robot;
	if(!arc) return;

	robot = &arc->robot;

	robot->Comm.PT = 2000; // 2s  timeout

	robot->Comm.CoolerSensPull_PT = 500; // 0.5s  timer

    robot->Comm.ArcComTimer.PT = robot->Comm.PT;

	if (robot->Comm.HeartBeat_Received && (robot->Comm.ArcComTimer.ET > 0)) //everytime got heartbeat, reset timer, to prevent trigger timeout
	    robot->Comm.ArcComTimer.IN = 0;

	else if (robot->Comm.HeartBeat_Received && (robot->Comm.ArcComTimer.ET == 0)){ //start timer, reset heartbeat flag
		if (robot->isMapped){  //
			robot->Comm.ArcComTimer.IN = 1;
		}
		if (robot->Comm.ClearError)    // clear error once getting connectivity from PS
		{
			robot->Comm.ClearError = 0;
			robot->Cntrl.Fbk.Error = 0;
			log_event(&robot->eventlog , "Network is active");
		}
		robot->Comm.HeartBeat_Received = 0;   //reset flag to start watchdog

	}

	TON(&robot->Comm.ArcComTimer);  //2 seconds Watchdog

    if (!robot->Comm.ArcComTimer.Q)
	robot->Comm.ArcLinkActive = 1;  // 1 Active
	else
	robot->Comm.ArcLinkActive = 0;	//timeout

	if (!robot->Comm.ArcLinkActive)
	{
		DBG_OB("Arc Link Disconnected\r\n");
		robot->Cntrl.Fbk.Error |= ArcLink_Com_Failed;
		robot->Cntrl.Fbk.Status = 0;
		robot->isMapping = 0;
		robot->isMapped = 0;	    //clear flag, set to unmapped status, stop timer
		robot->isMiscSetupOneShot = 0;
		robot->Comm.ArcComTimer.IN = 0;
		robot->Comm.ClearError = 1;	 //set flag when getting communication back, reset error
		log_event(&robot->eventlog , "Network is down");
	}
	else if (robot->isMapped)
	{
	/*	DBG_OB("Arc Link Connected\r\n"); */
		robot->Cntrl.Fbk.Error &= ~ArcLink_Com_Failed;
		robot->Cntrl.Fbk.Status |= ArcLink_Active;

	}

	// Pull Cooler Sens Status

	if((robot->miscSetup.CoolerAddr > 0)
		&& (robot->Comm.CoolerSensPull_PT > 0)){

		robot->Comm.CoolerSensPullTimer.PT = robot->Comm.CoolerSensPull_PT;

		if(robot->isMapped && robot->Comm.ArcLinkActive){

			if(!robot->Comm.CoolerSensPullTimer.IN){
				readAttribute_CoolerSens(arc);
				DBG("commanded Get Cooler Sens! \r\n" );
				robot->Comm.CoolerSensPullTimer.IN = 1;
				//TON(&robot->Comm.CoolerSensPullTimer);
			}
			else if(robot->Comm.CoolerSensPullTimer.Q){

				robot->Comm.CoolerSensPullTimer.IN = 0;
				//TON(&robot->Comm.CoolerSensPullTimer);

			}
			//else
				//TON(&robot->Comm.CoolerSensPullTimer);

		}

		TON(&robot->Comm.CoolerSensPullTimer);
	}

}
#endif /* _ROBOT_C */
```

### libUDP.c
```c
#ifdef _DEFAULT_INCLUDES
	#include <AsDefault.h>
#endif

/*
B&R components:
===============================================================================
*/
#include <bur/plc.h>
#include <bur/plctypes.h>

//void _NewDataSend(UDP_typ2* udp);

///////////////////////////////////////////////////////////////////////

 signed char Udp_cyclic(UDP_typ2* udp){

 	switch(udp->internal.step){

		case 0:

			udp->listener.oStatus.error_number = 0;
			udp->listener.oStatus.error = 0;
			udp->listener.oStatus.ready = 0;

			udp->send.oStatus.error_number = 0;
			udp->send.oStatus.error = 0;
			udp->send.oStatus.ready = 0;

			if(udp->listener_config.buffer && (udp->listener_config.bufferSize > 0)){

				if(udp->internal.UdpOpen_0.ident){ // CLose existing connection on start

					UdpClose(&udp->internal.UdpClose_0);  //Call the Function

					if(udp->internal.UdpClose_0.status == ERR_OK) //
						udp->internal.step = 1;

					else if (udp->internal.UdpClose_0.status == ERR_FUB_BUSY){} //UdpSend not finished -> redo

					else{  //Error

						udp->listener.oStatus.error_number = udp->internal.UdpClose_0.status;
						udp->listener.oStatus.error = 1;
						udp->listener.oStatus.ready = 0;
						udp->internal.step = 100;

					}

				}
				else
					udp->internal.step = 1;

			}
			else{ // No buffer declare

					udp->listener.oStatus.error_number = 0xFFFFF;
					udp->listener.oStatus.error = 1;
					udp->listener.oStatus.ready = 0;
					udp->internal.step = 100;

			}

		break;

		case 1:

			udp->internal.UdpOpen_0.enable = 1;

			if(udp->listener_config.ipAddress){

				if(strlen(udp->listener_config.ipAddress) >= 8 )
					udp->internal.UdpOpen_0.pIfAddr = udp->listener_config.ipAddress;
				else
					udp->internal.UdpOpen_0.pIfAddr = 0; // Listen to all addrresses

			}else
				udp->internal.UdpOpen_0.pIfAddr = 0; // Listen to all addrresses

			udp->internal.UdpOpen_0.port = udp->listener_config.port;	// Port to listen
			udp->internal.UdpOpen_0.options = 0;

			UdpOpen(&udp->internal.UdpOpen_0);	// Call the Function

			if(udp->internal.UdpOpen_0.status == ERR_OK
				|| udp->internal.UdpOpen_0.status == udpERR_ALREADY_EXIST){ // UdpOpen successful

				udp->internal.UdpSend_0.enable = 1;
				udp->internal.UdpSend_0.ident = udp->internal.UdpOpen_0.ident;	//Connection Ident from AsUDP.UDP_Open
				udp->internal.UdpSend_0.flags = 0;
				//
				udp->internal.UdpRecv_0.enable = 1;
				udp->internal.UdpRecv_0.ident = udp->internal.UdpOpen_0.ident;  //Connection Ident from AsUDP.UDP_Open
				udp->internal.UdpRecv_0.pData	= udp->listener_config.buffer;  // Where to store the incoming data
				udp->internal.UdpRecv_0.datamax = udp->listener_config.bufferSize;  // Lenght of data buffer
				udp->internal.UdpRecv_0.flags = 0;
				//
				udp->internal.UdpClose_0.enable = 1;
				udp->internal.UdpClose_0.ident = udp->internal.UdpOpen_0.ident;  //Connection Ident from AsUDP.UDP_Open
				//
				udp->listener.oStatus.ready = 1;
				udp->send.oStatus.ready = 1;
				udp->internal.step = 5;

			}
			else if( udp->internal.UdpOpen_0.status == ERR_FUB_BUSY ){}// UdpOpen not finished -> redo

			else {

				udp->listener.oStatus.error_number = udp->internal.UdpOpen_0.status;
				udp->listener.oStatus.error = 1;
				udp->listener.oStatus.ready = 0;
				udp->internal.step = 100;

			}

		break;

		case 5: // Receive Data from the PS and Trasmit to the PS

			UdpRecv(&udp->internal.UdpRecv_0);  // Call the Function

			if(udp->internal.UdpRecv_0.status == ERR_OK){// new response received

				udp->listener.oStatus.error = 0;
				udp->listener.oStatus.ready = 1;
				udp->listener.oDataLen = udp->internal.UdpRecv_0.recvlen;
				udp->listener.oStatus.counts++;

				if(udp->listener.iRxCallback){

					void (*rxCallback)(UDINT pBuf, UDINT LenData , UDINT ringBuf) =  ( void(*) (UDINT, UDINT , UDINT) ) udp->listener.iRxCallback;
					(*rxCallback)( (UDINT)udp->listener_config.buffer , udp->listener.oDataLen , udp->listener.iRxRingBuf);

				}

			}
			else if (udp->internal.UdpRecv_0.status == ERR_FUB_BUSY){} //UdpSend not finished -> redo

			else if (udp->internal.UdpRecv_0.status == udpERR_NO_DATA){} //UdpSend not finished -> redo

			else{

				udp->listener.oStatus.error_number = udp->internal.UdpRecv_0.status;
				udp->listener.oStatus.error = 1;
				udp->listener.oStatus.ready = 0;
				udp->internal.step = 100;

			}

		break;

		case 100:  // Error State

			if(udp->ResetCmd){
				udp->ResetCmd = 0;

				udp->internal.step ++;

			}

		break;

		case 200:  // Idle for test purpose

		break;

		default:

			udp->internal.step = 0;

		break;

	}

	_NewDataSend(udp);

	return 0;
 }

void _NewDataSend(UDP_typ2* udp){

	//////////////////////////////////////////////
	if(udp->send.iSendCMD){

		udp->listener.oStatus.error = 0;

		if(udp->internal.step == 5){ // UDP Opened

			udp->internal.UdpSend_0.pHost = udp->send.iIPaddress;
			udp->internal.UdpSend_0.port = udp->send.iPort;
			udp->internal.UdpSend_0.pData = udp->send.iBuffer;	// Which data to send
			udp->internal.UdpSend_0.datalen = udp->send.iBufferSize;	// data length

			UdpSend(&udp->internal.UdpSend_0);

			if(udp->internal.UdpSend_0.status == ERR_OK){// new data sent

				udp->send.iSendCMD = 0;
				udp->send.oStatus.counts++;

				if(udp->send.iTxCallback){

					void (*txCallback)(UDINT pBuf, UDINT LenData) =  ( void(*) (UDINT, UDINT) ) udp->send.iTxCallback;
					//(*txCallback)( (UDINT)udp->send.iBuffer , udp->send.iBufferSize );
					(*txCallback)( (UDINT)udp->internal.UdpSend_0.pData , udp->internal.UdpSend_0.sentlen);

				}

			}
			else if (udp->internal.UdpSend_0.status == ERR_FUB_BUSY){} //UdpSend not finished -> redo

			else{  //Error

				udp->send.iSendCMD = 0;

				udp->listener.oStatus.error_number = udp->internal.UdpRecv_0.status;
				udp->listener.oStatus.error = 1;

			}

		}
		else{ // Command error

			udp->send.iSendCMD = 0;

			udp->listener.oStatus.error_number = 0xFFFF;
			udp->listener.oStatus.error = 1;

		}

	}

}
```

### libUDP.h
```c
/* Automation Studio generated header file */
/* Do not edit ! */
/* libUDP  */

#ifndef _LIBUDP_
#define _LIBUDP_

/* Datatypes and datatypes of function blocks */
typedef struct Udp_Internal_typ
	{	unsigned char step;
	struct UdpOpen UdpOpen_0;
	struct UdpSend UdpSend_0;
	struct UdpRecv UdpRecv_0;
	struct UdpClose UdpClose_0;
} Udp_Internal_typ;

typedef struct Udp_Status_typ
	{	unsigned short error_number;
	plcbit error;
	plcbit ready;
	unsigned char counts;
} Udp_Status_typ;

typedef struct Udp_Config_typ
	{	plcstring ipAddress[21];
	unsigned short port;
	unsigned long bufferSize;
	signed char* buffer;
} Udp_Config_typ;

typedef struct Udp_Listener_Intrf_typ
	{	struct Udp_Status_typ oStatus;
	unsigned long oDataLen;
	unsigned long iRxCallback;
	unsigned long iRxRingBuf;
} Udp_Listener_Intrf_typ;

typedef struct Udp_Send_Intrf_typ
	{	struct Udp_Status_typ oStatus;
	plcbit iSendCMD;
	plcstring iIPaddress[21];
	unsigned short iPort;
	unsigned long iBufferSize;
	signed char* iBuffer;
	unsigned long iTxCallback;
} Udp_Send_Intrf_typ;

typedef struct UDP_typ2
	{	struct Udp_Listener_Intrf_typ listener;
	struct Udp_Send_Intrf_typ send;
	struct Udp_Config_typ listener_config;
	struct Udp_Internal_typ internal;
	plcbit ResetCmd;
} UDP_typ2;

#endif /* _LIBUDP_ */
```

Listed in the project but not available here: Logical/Global.typ, Logical/Global.var, Logical/IO/Types.typ, Logical/IO/Variables.var, Logical/UDP/Types.typ, Logical/IndexMtr/Types.typ, Logical/IndexMtr/Variables.var, Logical/TcpCam/Types.typ, Logical/TcpCam/bgsprintf.c, Logical/TcpCam/bgsprintf.h, Logical/TML_Cfg/Types.typ, Logical/TML_Cfg/Variables.var, Logical/MainProc/Types.typ, Logical/MainProc/Variables.var, Logical/BR_Modbus/Types.typ, Logical/BR_Modbus/Variables.var, Logical/Calibr/Types.typ, Logical/Calibr/Variables.var, Logical/LocalJog/Types.typ, Logical/LocalJog/Variables.var, Logical/Tester/Types.typ, Logical/Tester/Variables.var, Logical/HMI_Report/Types.typ, Logical/HMI_Report/Variables.var, Logical/Lib/DataMgrLib.c, Logical/Lib/DataMgrLib.h, Logical/Lib/statelib.h, Logical/Lib/xstring.h, Logical/Lib/utilityLib/bgringbuffer.c, Logical/Lib/utilityLib/bgringbuffer.h, Logical/Lib/utilityLib/bgsprintf.c, Logical/Lib/utilityLib/bgsprintf.h, Logical/Lib/utilityLib/bgstring.c, Logical/Lib/utilityLib/bgstring.h, Logical/Lib/utilityLib/libRingBuffer.c, Logical/Lib/utilityLib/libRingBuffer.h, Logical/Lib/arclink/NetworkAttribute.h, Logical/Lib/arclink/WeldController.h, Logical/Lib/arclink/NetworkBlocks.h, Logical/Lib/arclink/ArcLinkObject.h, Logical/Lib/arclink/ArcLinkMap.h, Logical/Lib/arclink/Attribute.h, Logical/Lib/arclink/MessageBuilder.c, Logical/Lib/arclink/ArcLinkMap.c, Logical/Lib/arclink/IncomingHandler.c, Logical/Lib/arclink/NetworkActions.h, Logical/Lib/arclink/WeldController.c, Logical/Lib/arclink/ArcLinkUtility.c, Logical/Lib/arclink/Robot.h
